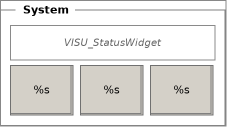
VISUALIZATION VISU_SystemControl  // 227x127
VAR_IN_OUT
    status : StatusWidget;
	button_initialize : InitializeButtonWidget;
    button_operating : OperatingButtonWidget;
    button_locking : LockingButtonWidget;
END_VAR
    Polyline (15,10) (0,10) (0,125) (225,125) (225,10) (75,10)
    Button (150,65 63x50), "%s", text variable: button_operating.text, input disabled if: button_operating.deactivate
        OnMouseClick: execute { button_operating.do_request := TRUE; }
    Button (80,65 63x50), "%s", text variable: button_locking.text, input disabled if: button_locking.deactivate
        OnMouseClick: execute { button_locking.do_request := TRUE; }
    Frame (10,25 205x35)
        shows VISU_StatusWidget(widget := status)
    Button (10,65 63x50), "%s", text variable: button_initialize.text, input disabled if: button_initialize.deactivate
        OnMouseClick: execute { button_initialize.do_request := TRUE; }
    Label (20,0 55x20), "System"
END_VISUALIZATION

(* stored: Version 1.1.0.1, ProductVersion 3.1.4019.2
   Visu VISU_SystemControl: Id {aa485310-71c0-4c56-a921-d869ce425eed} *)
